DATA_BLOCK "PN-INOUT14"
{ S7_Optimized_Access := 'FALSE' }
VERSION : 0.1
   STRUCT
      a01 : Byte;
      b01 : Byte;   // DO_BYTE1 захват команды
      c01 : Byte;   // DO_BYTE2 состояния
      d01 : Byte;   // DO_BYTE3 ошибки
      e01 : Byte;   // DO_BYTE4 UO
      f01 : Byte;   // DO_BYTE5 Текущий ряд, линия 1
      g01 : Byte;   // DO_BYTE6 Позиция в ряду, линия 1
      h01 : Byte;   // DO_BYTE7 Текущий ряд, линия 2
      i01 : Byte;   // DO_BYTE8 Позиция в ряду, линия 2
      J01 : Byte;   // DO_BYTE9 Моточасы1
      K01 : Byte;   // DO_BYTE10 Моточасы2
      L01 : Byte;
      M01 : Byte;
      N01 : Byte;
      O01 : Byte;
      P01 : Byte;
      Q01 : Byte;
      R01 : Byte;   // DI_BYTE1 датчики захвата
      S01 : Byte;   // DI_BYTE2 датчики паллет
      T01 : Byte;   // DI_BYTE3 присоски
      a2 : Byte;   // DI_BYTE4 UI
      b2 : Byte;   // DI_BYTE5 Скорость робота
      c2 : Byte;
      d2 : Byte;
      e2 : Byte;
      f2 : Byte;
      g2 : Byte;
      h2 : Byte;
      i2 : Byte;
      J2 : Byte;
      K2 : Byte;
      L2 : Byte;
      M2 : Byte;
      N2 : Byte;
      O2 : Byte;
      P2 : Byte;
      Q2 : Byte;
      R2 : Byte;
      S2 : Byte;
      T2 : Byte;
   END_STRUCT;


BEGIN

END_DATA_BLOCK

